FUNCTION_BLOCK FB_addReal
VAR_INPUT
END_VAR
VAR_OUTPUT
END_VAR
VAR
END_VAR

END_FUNCTION_BLOCK

(* stored: Version 1.1.0.1, ProductVersion 3.1.4024.12
   POU FB_addReal: Id {44fe6edb-c9c1-40ba-a757-3d7869c99e5f}, SpecialFunc None *)
